Yaskawa INFORM job: AVANCA_PINOS.JBI

/JOB
//NAME AVANCA_PINOS
///FOLDERNAME GRAMPOS
//POS
///NPOS 0,0,0,0,0,0
//INST
///DATE 2022/06/09 09:52
///ATTR SC,RW
NOP
DOUT OT#(540) OFF
DOUT OT#(539) ON
WAIT IN#(546)=ON
WAIT IN#(548)=ON
END
